// TIA Portal project "TSI_LI_safety" (V15.1)

(* hardware
DEVICE "S71500/ET200MP station_1"  S7-1500 station
   slot 0: "Rail_0"  Rack  6ES7 590-1***0-0AA0
   slot 1: "PLC_1"  CPU 1516F-3 PN/DP  6ES7 516-3FN00-0AB0  V1.8
      slot 3: "CPU display_1"  6ES7591-1BA00-0AA0
DEVICE "ET 200SP station_1"  ET 200SP-Station
   slot 0: "Rack_0"  Rack  6ES5 710-8MAx1
   slot 0: "120ET2"  IM 155-6 PN HF  6ES7 155-6AU00-0CN0  V4.2
   slot 1: "121DI0"  F-DI 8x24VDC HF  6ES7 136-6BA00-0CA0  V1.0
      slot 1: "121DI0"  F-DI 8x24VDC HF
   slot 2: "123DI0"  DI 8x24VDC BA  6ES7 131-6BF00-0AA0  V1.0
      slot 1: "123DI0"  DI 8x24VDC BA
   slot 3: "124DI0"  DI 8x24VDC BA  6ES7 131-6BF00-0AA0  V1.0
      slot 1: "124DI0"  DI 8x24VDC BA
   slot 4: "125AI0"  AI 2xU ST  6ES7 134-6FB00-0BA1  V1.0
      slot 1: "125AI0"  AI 2xU ST
   slot 5: "Server module_1"  Server module  6ES7 193-6PA00-0AA0  V1.1
      slot 1: "Server module_1"  Server module
   slot 127: "BA 2xRJ45"  BA 2xRJ45  6ES7 193-6AR00-0AA0  V0.0
      slot 1: "Port_1"  X1 P1 R  6ES7 193-6AR00-0AA0  V0.0
      slot 2: "Port_2"  X1 P2 R  6ES7 193-6AR00-0AA0  V0.0
DEVICE "ET 200SP station_2"  ET 200SP-Station
   slot 0: "Rack_0"  Rack  6ES5 710-8MAx1
   slot 0: "220ET2"  IM 155-6 PN HF  6ES7 155-6AU00-0CN0  V4.2
   slot 1: "202DI0"  F-DI 8x24VDC HF  6ES7 136-6BA00-0CA0  V1.0
      slot 1: "202DI0"  F-DI 8x24VDC HF
   slot 2: "204DI0"  DI 8x24VDC ST  6ES7 131-6BF00-0BA0  V1.1
      slot 1: "204DI0"  DI 8x24VDC ST
   slot 3: "205DI0"  DI 8x24VDC ST  6ES7 131-6BF00-0BA0  V1.1
      slot 1: "205DI0"  DI 8x24VDC ST
   slot 4: "206FPM2"  F-PM-E 24VDC/8A PPM ST  6ES7 136-6PA00-0BC0  V2.0
      slot 1: "206FPM2"  F-PM-E 24VDC/8A PPM ST
   slot 5: "207DO0"  DQ 8x24VDC/0.5A ST  6ES7 132-6BF00-0BA0  V1.1
      slot 1: "207DO0"  DQ 8x24VDC/0.5A ST
   slot 6: "Server module_1"  Server module  6ES7 193-6PA00-0AA0  V1.1
      slot 1: "Server module_1"  Server module
   slot 127: "BA 2xRJ45"  BA 2xRJ45  6ES7 193-6AR00-0AA0  V0.0
      slot 1: "Port_1"  X1 P1 R  6ES7 193-6AR00-0AA0  V0.0
      slot 2: "Port_2"  X1 P2 R  6ES7 193-6AR00-0AA0  V0.0
*)

// ===== PLC "PLC_1"  CPU 1516F-3 PN/DP =====
// protected blocks, not shown: "Main_Safety_RTG1", "Main_Safety_RTG1_DB"

VAR_GLOBAL   // PLC tag table "Default tag table"
   "E-Stop_Stand" AT %I12.0 : Bool;   // Emergancy stop (Measuring stand)
   "SICK" AT %I12.1 : Bool;   // SICK sensor
   "Robot_ON" AT %I12.3 : Bool;   // Robot ON relay callback
   "E-Stop_MC" AT %I0.0 : Bool;   // Emergancy STOP main cabinet
   "PM_switch" AT %Q20.0 : Bool;   // Power module output control
   "Robot output" AT %Q4.0 : Bool;
END_VAR

DATA_BLOCK "TSI_LI_Datablock"   // DB2
{ S7_Optimized_Access := 'TRUE' }
VERSION : 0.1
   VAR
      Safety_ACK : Bool;   // Safety ack button WinCC
      Robot_Output_Check : Bool;
      VstupET1 : Bool;
      VstupET2 : Bool;
   END_VAR
BEGIN
END_DATA_BLOCK

ORGANIZATION_BLOCK "Main"   // OB1, LAD, ProgramCycle
TITLE = "Main Program Sweep (Cycle)"
{ S7_Optimized_Access := 'TRUE' }
VERSION : 0.1
   VAR_INPUT
      Initial_Call : Bool;   // Initial call of this OB
      Remanence : Bool;   // =True, if remanent data are available
   END_VAR
   VAR_TEMP
      Out : Bool;
   END_VAR
BEGIN
END_ORGANIZATION_BLOCK